PROGRAM P4_06_DiskSize
VAR
	fbSize				:FB_PythonScript;
	rFreeSpacePer		:REAL;
	bLowSpace			:BOOL;
END_VAR

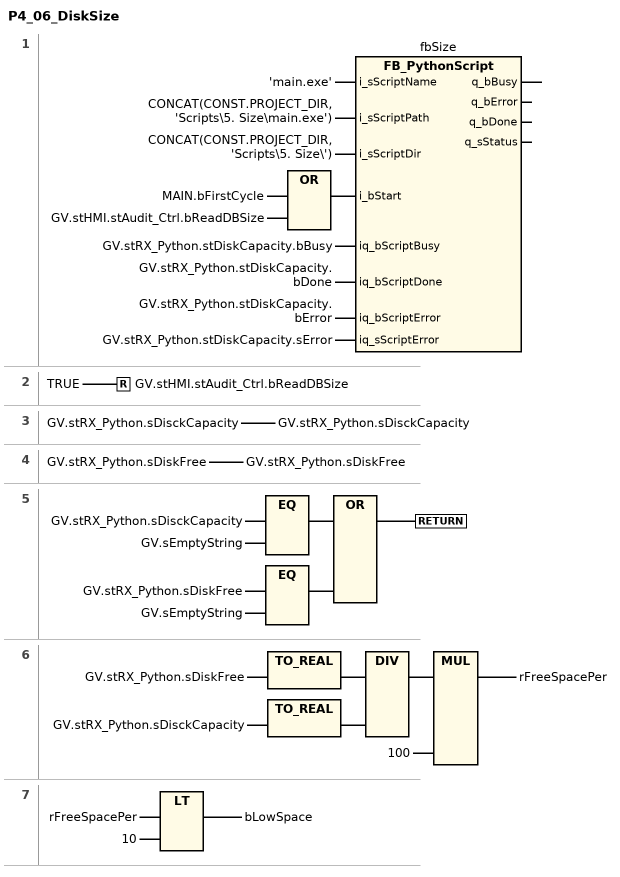
// NETWORK 1
fbSize(
    i_sScriptName := 'main.exe',
    i_sScriptPath := CONCAT(CONST.PROJECT_DIR,'Scripts\5. Size\main.exe'),
    i_sScriptDir := CONCAT(CONST.PROJECT_DIR,'Scripts\5. Size\'),
    i_bStart := MAIN.bFirstCycle OR GV.stHMI.stAudit_Ctrl.bReadDBSize,
    iq_bScriptBusy := GV.stRX_Python.stDiskCapacity.bBusy,
    iq_bScriptDone := GV.stRX_Python.stDiskCapacity.bDone,
    iq_bScriptError := GV.stRX_Python.stDiskCapacity.bError,
    iq_sScriptError := GV.stRX_Python.stDiskCapacity.sError); // FB_PythonScript

// NETWORK 2
GV.stHMI.stAudit_Ctrl.bReadDBSize R= TRUE;

// NETWORK 3
GV.stRX_Python.sDisckCapacity := GV.stRX_Python.sDisckCapacity;

// NETWORK 4
GV.stRX_Python.sDiskFree := GV.stRX_Python.sDiskFree;

// NETWORK 5
IF GV.stRX_Python.sDisckCapacity = GV.sEmptyString OR GV.stRX_Python.sDiskFree = GV.sEmptyString THEN RETURN; END_IF

// NETWORK 6
rFreeSpacePer := (TO_REAL(GV.stRX_Python.sDiskFree) / TO_REAL(GV.stRX_Python.sDisckCapacity)) * 100;

// NETWORK 7
bLowSpace := rFreeSpacePer < 10;

END_PROGRAM

(* stored: Version 1.1.0.1, ProductVersion 3.1.4024.12
   POU P4_06_DiskSize: Id {37c73627-27c3-4fae-9810-f82ba81eb48e}, SpecialFunc None *)
